Staubli VAL3: moveZero.pgx

program moveZero()
begin
  movej(zeroPosition,flange,mFastMov)
  waitEndMove()
  message="moveZero:done"
  taskCreate "sendStatus",100,sendStatus()
  taskKill("moveZero")
end
